TYPE ChangeSetpointProcessArgs :
STRUCT
	///New setpoint value
	setpoint: LREAL;
END_STRUCT
END_TYPE

(* stored: Version 1.1.0.1, ProductVersion 3.1.4019.2
   DUT ChangeSetpointProcessArgs: Id {2317f587-cf95-459a-be1e-e174404ee134} *)
